# EPICS substitutions: lsredis/iocBoot/iocLinux/async_pid_slow.substitutions
# This file demonstrates slow feedback.  The initial INP and OUT assume the first channel
# of an IP330 ADC connected to the first channel of a DAC128V DAC.
file "$(STD)/stdApp/Db/async_pid_control.db"
{
pattern
{P,      PID,              INP,        OUT, LOPR,   HOPR,  DRVL, DRVH,  PREC,      KP,  KI,   KD,  SCAN}
{lsredis:,   async_pid_slow, lsredis:userCalcOut10, lsredis:userCalcOut10.A,    0,    100,     0,    5,     3,     0.2,  3.,   0.,  ".1 second"}
}
